RoboDK station: Stringer B-Top1-BOX2.rdk

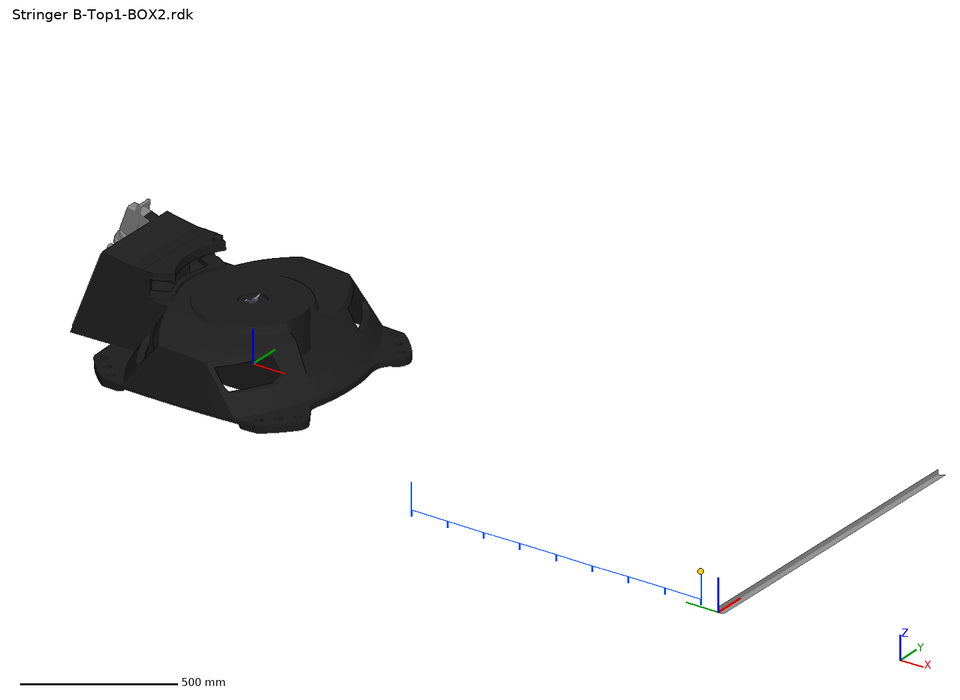
[picture v0: the station drawn from its stored meshes, robots at their saved joint values, targets as dots, program paths as lines]
Station Stringer B-Top1-BOX2 (saved by RoboDK 5.2.3). Poses are relative to the parent item; angles as X-Y-Z fixed-axis rotations.
  - frame KUKA KR 210 R2700 extra Base at (0, 0, 0) mm
    - robot KUKA KR 210 R2700 extra: 6 axes, payload 210 kg, reach 2696 mm, repeatability 0.06 mm, weight 1068 kg
        joint limits [-185, -140, -120, -350, -125, -350] to [185, -5, 155, 350, 125, 350]; home [0, -90, 90, 0, 0, 0]; saved at [-37.863, -26.817, 86.564, 95.563, 22.835, -127.172]
      - tool Spindle, TCP at (32, 0, 260) mm, rotated rx 0 ry 39 rz 0 deg, size 157.3 x 72 x 259.9 mm
  - frame Frame 2 at (1800, 0, -372.68) mm, rotated rx 0 ry 0 rz 90 deg
    - object L-Stringer B - Top1-BOX2 at (0, 0, 0) mm, rotated rx 90 ry 0 rz 0 deg, size 1223.8 x 20 x 20 mm, geometry from L-Stringer B - Top1-BOX2.stl
    - object Stringer B-Top1-BOX2 at (0, 0, 0) mm, rotated rx 0 ry 0 rz -90 deg, 9 curves, geometry from Point 9
  - machining project Point settings: rotZ(0) | rotX(0)*rotY(0) | rotz(0) | onStart | onPathStart | onApproach | onPoint | onRetract | onFinish | SetRPM(%1) | SetTool(%1) | Extruder(%1) | default | default | OutOnMov(%1) | OutOffMov(%1) | onPathFinish | M_RunCode(%1)
  - program Point (56 instructions, listed below)
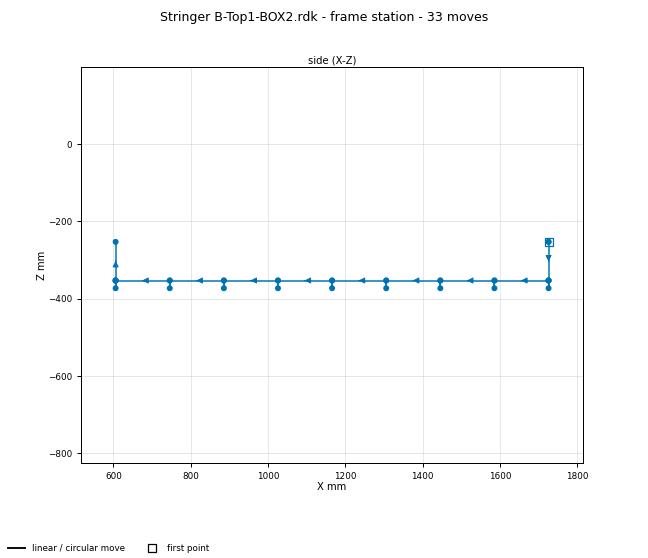
[picture p0: tool path of Stringer B-Top1-BOX2.rdk in frame station, 33 of 33 moves have a stored position in this frame; points joined in program order, loops and branches not executed]

--- program Point (robot KUKA KR 210 R2700 extra) ---
  Smooth(1)
  Set speed (1000.0 mm/s)
  Set Ref.: Frame 2
  Set Tool: Spindle
  Show Spindle
  MoveJ 1 to (10, 73.93, 120) mm, rotated rx 180 ry 0 rz -180 deg; joints [-2.756, -33.796, 110.696, 176.031, 25.922, -178.572]
  MoveL 2 to (10, 73.93, 120) mm, rotated rx 180 ry 0 rz -180 deg; joints [-2.756, -33.796, 110.696, 176.031, 25.922, -178.572]
  MoveL 3 to (10, 73.93, 20) mm, rotated rx 180 ry 0 rz 180 deg; joints [-2.756, -28.523, 108.075, 176.372, 28.567, -178.955]
  MoveL 4 to (10, 73.93, 20) mm, rotated rx 180 ry 0 rz 180 deg; joints [-2.756, -28.523, 108.075, 176.372, 28.567, -178.955]
  Set speed (50.0 mm/s)
  MoveL 5 to (10, 73.93, 0) mm, rotated rx 180 ry 0 rz 180 deg; joints [-2.756, -27.475, 107.503, 176.427, 29.042, -179.017]
  MoveL 6 to (10, 73.93, 20) mm, rotated rx 180 ry 0 rz 180 deg; joints [-2.756, -28.523, 108.075, 176.372, 28.567, -178.955]
  Set speed (1000.0 mm/s)
  MoveL 7 to (10, 213.95, 20) mm, rotated rx 180 ry 0 rz -180 deg; joints [-7.93, -28.418, 107.388, 169.381, 28.11, -176.789]
  Set speed (50.0 mm/s)
  MoveL 8 to (10, 213.95, 0) mm, rotated rx 180 ry 0 rz -180 deg; joints [-7.93, -27.376, 106.818, 169.542, 28.575, -176.971]
  MoveL 9 to (10, 213.95, 20) mm, rotated rx 180 ry 0 rz -180 deg; joints [-7.93, -28.418, 107.388, 169.381, 28.11, -176.789]
  Set speed (1000.0 mm/s)
  MoveL 10 to (10, 353.97, 20) mm, rotated rx 180 ry 0 rz 180 deg; joints [-12.978, -28.194, 106.036, 162.033, 27.269, -174.075]
  Set speed (50.0 mm/s)
  MoveL 11 to (10, 353.97, 0) mm, rotated rx 180 ry 0 rz -180 deg; joints [-12.978, -27.163, 105.471, 162.307, 27.712, -174.384]
  MoveL 12 to (10, 353.97, 20) mm, rotated rx 180 ry 0 rz 180 deg; joints [-12.978, -28.194, 106.036, 162.033, 27.269, -174.075]
  Set speed (1000.0 mm/s)
  MoveL 13 to (10, 493.99, 20) mm, rotated rx 180 ry 0 rz -180 deg; joints [-17.829, -27.823, 104.025, 154.08, 26.156, -170.465]
  Set speed (50.0 mm/s)
  MoveL 14 to (10, 493.99, 0) mm, rotated rx 180 ry 0 rz 180 deg; joints [-17.829, -26.809, 103.467, 154.479, 26.565, -170.91]
  MoveL 15 to (10, 493.99, 20) mm, rotated rx 180 ry 0 rz -180 deg; joints [-17.829, -27.823, 104.025, 154.08, 26.156, -170.465]
  Set speed (1000.0 mm/s)
  MoveL 16 to (10, 634.01, 20) mm, rotated rx -180 ry 0 rz -180 deg; joints [-22.43, -27.269, 101.362, 145.274, 24.931, -165.636]
  Set speed (50.0 mm/s)
  MoveL 17 to (10, 634.01, 0) mm, rotated rx -180 ry 0 rz -180 deg; joints [-22.43, -26.275, 100.81, 145.807, 25.295, -166.224]
  MoveL 18 to (10, 634.01, 20) mm, rotated rx -180 ry 0 rz -180 deg; joints [-22.43, -27.269, 101.362, 145.274, 24.931, -165.636]
  Set speed (1000.0 mm/s)
  MoveL 19 to (10, 774.03, 20) mm, rotated rx 180 ry 0 rz -180 deg; joints [-26.746, -26.49, 98.05, 135.411, 23.793, -159.338]
  Set speed (50.0 mm/s)
  MoveL 20 to (10, 774.03, 0) mm, rotated rx 180 ry 0 rz -180 deg; joints [-26.746, -25.52, 97.504, 136.078, 24.097, -160.068]
  MoveL 21 to (10, 774.03, 20) mm, rotated rx 180 ry 0 rz -180 deg; joints [-26.746, -26.49, 98.05, 135.411, 23.793, -159.338]
  Set speed (1000.0 mm/s)
  MoveL 22 to (10, 914.05, 20) mm, rotated rx 180 ry 0 rz -180 deg; joints [-30.757, -25.446, 94.085, 124.427, 22.965, -151.484]
  Set speed (50.0 mm/s)
  MoveL 23 to (10, 914.05, 0) mm, rotated rx 180 ry 0 rz -180 deg; joints [-30.757, -24.5, 93.544, 125.207, 23.197, -152.332]
  MoveL 24 to (10, 914.05, 20) mm, rotated rx 180 ry 0 rz -180 deg; joints [-30.757, -25.446, 94.085, 124.427, 22.965, -151.484]
  Set speed (1000.0 mm/s)
  MoveL 25 to (10, 1054.07, 20) mm, rotated rx 180 ry 0 rz 180 deg; joints [-34.461, -24.092, 89.453, 112.52, 22.674, -142.269]
  Set speed (50.0 mm/s)
  MoveL 26 to (10, 1054.07, 0) mm, rotated rx -180 ry 0 rz -180 deg; joints [-34.461, -23.171, 88.915, 113.36, 22.823, -143.181]
  MoveL 27 to (10, 1054.07, 20) mm, rotated rx 180 ry 0 rz 180 deg; joints [-34.461, -24.092, 89.453, 112.52, 22.674, -142.269]
  Set speed (1000.0 mm/s)
  MoveL 28 to (10, 1194.09, 20) mm, rotated rx -180 ry 0 rz -180 deg; joints [-37.863, -22.384, 84.119, 100.212, 23.109, -132.221]
  Set speed (50.0 mm/s)
  MoveL 29 to (10, 1194.09, 0) mm, rotated rx 180 ry 0 rz -180 deg; joints [-37.863, -21.487, 83.58, 101.034, 23.175, -133.115]
  MoveL 30 to (10, 1194.09, 20) mm, rotated rx -180 ry 0 rz -180 deg; joints [-37.863, -22.384, 84.119, 100.212, 23.109, -132.221]
  MoveL 31 to (10, 1194.09, 20) mm, rotated rx -180 ry 0 rz -180 deg; joints [-37.863, -22.384, 84.119, 100.212, 23.109, -132.221]
  Set speed (1000.0 mm/s)
  MoveL 32 to (10, 1194.09, 20) mm, rotated rx -180 ry 0 rz -180 deg; joints [-37.863, -22.384, 84.119, 100.212, 23.109, -132.221]
  MoveL 33 to (10, 1194.09, 120) mm, rotated rx 180 ry 0 rz -180 deg; joints [-37.863, -26.817, 86.564, 95.563, 22.835, -127.172]
